TYPE ST_LaudaReadCommands_Safety :
STRUCT
	CommTimeoutViaInterface : STRING := 'IN_SP_08';
	SafetyModeActive		: STRING := 'IN_MODE_06';
END_STRUCT
END_TYPE

(* stored: Version 1.1.0.1, ProductVersion 3.1.4024.12
   DUT ST_LaudaReadCommands_Safety: Id {f348e1ff-c058-4094-86f4-14f86470224c} *)
